FUNCTION_BLOCK Sensor_Model
  (* Version 0.1, 2005-12-13, Oscar Ljungkrantz, Chalmers *)
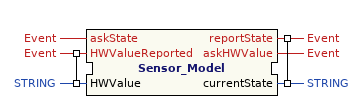
  EVENT_INPUT
    askState;
    HWValueReported WITH HWValue;
  END_EVENT
  EVENT_OUTPUT
    reportState WITH currentState;
    askHWValue;
  END_EVENT
  VAR_INPUT
    HWValue : STRING;
  END_VAR
  VAR_OUTPUT
    currentState : STRING;
  END_VAR
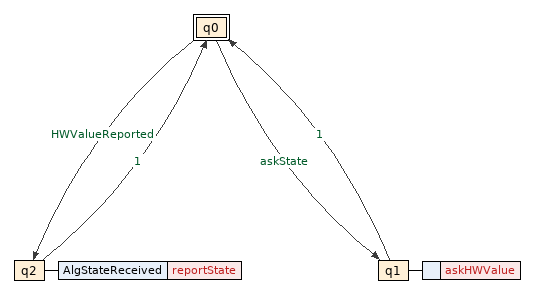
  EC_STATES
    q0;
    q1 : -> askHWValue;
    q2 : AlgStateReceived -> reportState;
  END_STATES
  EC_TRANSITIONS
    q0 TO q1 := askState;
    q0 TO q2 := HWValueReported;
    q1 TO q0 := 1;
    q2 TO q0 := 1;
  END_TRANSITIONS
  ALGORITHM AlgStateReceived IN Java:
currentState = HWValue;
  END_ALGORITHM
END_FUNCTION_BLOCK
(* other elements stored in the file *)
(* InternalVars> <VarDeclaration Name="" Type="" InitialValue="" /> </InternalVars *)
